(* PLC project PRINCIPAL, Beckhoff Automation GmbH TwinCAT PLC Control 3.5.13.21 *)
(* stored: creationDateTime 2022-11-03T11:03:07.8325215, modificationDateTime 2022-11-03T11:03:07.8345215 *)

PROGRAM pConfig_Control
VAR_INPUT
END_VAR
VAR_OUTPUT
END_VAR
VAR
	ActvHorn: fHorn;
	TestSirena: BOOL;
END_VAR

            (*-------------------------------------------------------------------------------------------------------*)
(*-------------------------------------------------------------------------------------------------------*)
(*CARGA PF*)
Mc.CONTROL.iPFTempAlta:= WORD_TO_INT(PF[2]);			(*Temperatura para marcar temperatua alta*)


(*-------------------------------------------------------------------------------------------------------*)
(*Pulsadores auto man*)
ATL.PE.xPulAuto := Mc.CONTROL.p401_PAuto.bPul;
ATL.PE.xPulMan := Mc.CONTROL.p400_PMAn.bPul;
Mc.CONTROL.p400_PMAn.bPilot:= aTL.PE.xMan;
MC.CONTROL.p401_PAuto.bPilot:= ATL.PE.xAuto; 
 
(*-------------------------------------------------------------------------------------------------------*)
(*Gestion Alarmes*)
ActvHorn(
	axAlarm:= ATL.PE.axAlarm, 
	axHorn:= ATL.PE.axHorn, 
	xStopHorn:= ATL.PE_COM.xStopAlarm OR Mc.CONTROL.p402_StopAlarm.bPul, 
	);

Mc.CONTROL.xAlarmActv:= ActvHorn.xAlarmActv;
TestSirena := ActvHorn.xHornActv;

(*Maquina Caliente*)
IF Mc.CONTROL.iPFTempAlta>0
	THEN
	Mc.CONTROL.xMcHot:= (Mc.TEMP.rMacTemperature>Mc.CONTROL.iPFTempAlta);
	ELSE
	Mc.CONTROL.xMcHot:= Mc.SEG.xMaxPresTemp;
END_IF


(*Maquina Pausada*)
Mc.control.xMcPaused:= Mc.CONTROL.p407_Pause.bPul;




          
END_PROGRAM
